# B&R Automation Studio project mappFramework (part 12)

#### variables.var - Name the suite and add PVs for the program
```iecst
(********************************************************************
 * COPYRIGHT --
 ********************************************************************
 * Program: utTemplate_automated
 * File: variables.var
 * Author: -
 * Created: -
 ********************************************************************
 * Local variables of program utTemplate_automated
 ********************************************************************)
(*Describe the test*)
VAR
	Testsuite : UtMgrTestSuite := (Name:='RecipeMgrVC4',Description:='RecipeMgr VC4 Unit Tests',MetaInformation:='Meta');
END_VAR
(*Variables used in the tests*)
VAR
	cycleCount : {REDUND_UNREPLICABLE} USINT;
	pMachineSettings : REFERENCE TO MachineSettingsType;
	MachineSettingsSize : {REDUND_UNREPLICABLE} UDINT;
	pParameters : REFERENCE TO ParametersType;
	ParameterSize : {REDUND_UNREPLICABLE} UDINT;
	LastSelectedIndex : UDINT;
	SetupState : USINT;
	FileName : STRING[24];
	NumberOfFiles : UINT;
	CurrentFile : UINT;
	fileInfo : fiDIR_READ_DATA;
	DirInfo_UT : DirInfo;
	DirRead_UT : DirRead;
	FileDelete_UT : FileDelete;
	FileCopy_UT : FileCopy;
END_VAR
```

#### testSuite.h
```c
#ifndef __TEST_SUITE_H__
#define __TEST_SUITE_H__

bool RecipeExists(char* recipeName);
bool SelectRecipe(char* wantedRecipe);
testStatusEnum RemoveNonDefaultFiles(USINT categoryIndex, char* selectFile, const char* category);

#endif
```

#### testSuite.c
```c
/********************************************************************
 * COPYRIGHT --
 ********************************************************************
 * Program: -
 * Author:
 * Created:
 ********************************************************************
 * Test registration and handshake
 ********************************************************************/

#include <bur/plctypes.h>

#ifdef _DEFAULT_INCLUDES
#include <AsDefault.h>
#endif

#include "UnitTest.h"
#include <string.h>
#include <stdbool.h>

void _INIT initTestSuite(void)
{
	Testsuite.Enable = 1;
	utInit(&Testsuite);

	CommonTestsuite.Enable = 1;
	utInit(&CommonTestsuite);

	strcpy((char*)&FileDeviceName, "mappRecipeFiles");
	strcpy((char*)&TextNameSpace, "mappFramework/Recipe/Alarms");
	strcpy((char*)&TextID, "SaveFailed");
	strcpy((char*)&HmiRecipe.Parameters.DeviceName, "mappRecipeFiles");

	PV_xgetadr("RecipeMgr:MachineSettings", (void*)&pMachineSettings, &MachineSettingsSize);
	PV_xgetadr("RecipeMgr:Parameters", (void*)&pParameters, &ParameterSize);

	LastSelectedIndex++;
}

void _CYCLIC cyclicWithTest(void)
{
	utCyclic(&Testsuite);
	if (Testsuite.Informational.LastKnownPassedLocation.TestCaseName != 0)
		strcpy((char*)&LastTestCase, (char*)Testsuite.Informational.LastKnownPassedLocation.TestCaseName);
	if (Testsuite.Informational.LastKnownPassedLocation.TestSetName != 0)
		strcpy((char*)&LastTestSet, (char*)Testsuite.Informational.LastKnownPassedLocation.TestSetName);
	if (Testsuite.Informational.LastKnownPassedLocation.File != 0)
		strcpy((char*)&LastTestFile, (char*)Testsuite.Informational.LastKnownPassedLocation.File);
}

void _EXIT exitTestSuite(void)
{
	utExit(&Testsuite);
}

bool RecipeExists(char* recipeName)
{
	for (USINT i = 0; i<(sizeof(MpRecipeUIConnect.Recipe.List.Names)/sizeof(MpRecipeUIConnect.Recipe.List.Names[0])); i++)
	{
		if (strcmp(recipeName, MpRecipeUIConnect.Recipe.List.Names[i]) == 0)
		{
			return true;
		}
	}
	return false;
}

bool SelectRecipe(char* wantedRecipe)
{
	if (((MpRecipeUIConnect.Status != mpRECIPE_UI_STATUS_IDLE) && (MpRecipeUIConnect.Status != mpRECIPE_UI_STATUS_ERROR)) &&
		(strcmp(wantedRecipe, HmiRecipe.Status.SelectedRecipe) != 0)) return false;

	for (USINT i=0; i <= MpRecipeUIConnect.Recipe.List.MaxSelection; i++)
	{
		if (strcmp(wantedRecipe, MpRecipeUIConnect.Recipe.List.Names[i]) == 0)
			MpRecipeUIConnect.Recipe.List.SelectedIndex = i;
	}

	return (strcmp(wantedRecipe, HmiRecipe.Status.SelectedRecipe) == 0);
}

testStatusEnum RemoveNonDefaultFiles(USINT categoryIndex, char* selectFile, const char* category)
{
	switch (SetupState)
	{
		case 0:
			DirInfo_UT.enable = true;
			DirInfo_UT.pDevice = (UDINT)&"mappRecipeFiles";
			DirInfo_UT.pPath = (UDINT)&"";
			DirInfo(&DirInfo_UT);
			TEST_BUSY_CONDITION(DirInfo_UT.status == 65535);
			TEST_ABORT_CONDITION(DirInfo_UT.status != 0);
			NumberOfFiles = DirInfo_UT.filenum;
			CurrentFile = 0;
			SetupState = (NumberOfFiles == 0) ? 100 : 1;
			break;

		case 1:
			DirRead_UT.enable = true;
			DirRead_UT.pDevice = DirInfo_UT.pDevice;
			DirRead_UT.entry = CurrentFile;
			DirRead_UT.option = fiFILE;
			DirRead_UT.pData = (UDINT)&fileInfo;
			DirRead_UT.data_len = sizeof(fileInfo);
			DirRead(&DirRead_UT);
			TEST_BUSY_CONDITION(DirRead_UT.status == 65535);
			TEST_ABORT_CONDITION(DirRead_UT.status != 0);
			SetupState = 2;
			break;

		case 2:
			if ((strcmp("Default.par", (char*)fileInfo.Filename) == 0) ||
				(strcmp("Machine.mcfg", (char*)fileInfo.Filename) == 0))
			{
				CurrentFile++;
				SetupState = (CurrentFile >= NumberOfFiles) ? 10 : 1;
				break;
			}
			FileDelete_UT.enable = true;
			FileDelete_UT.pDevice = DirInfo_UT.pDevice;
			FileDelete_UT.pName = (UDINT)&fileInfo.Filename;
			FileDelete(&FileDelete_UT);
			TEST_BUSY_CONDITION(FileDelete_UT.status == 65535);
			TEST_ABORT_CONDITION(FileDelete_UT.status != 0);

			NumberOfFiles--;
			SetupState = (CurrentFile >= NumberOfFiles) ? 10 : 1;
			break;

		case 10:
			strcpy((char*)&HmiRecipe.Parameters.DeviceName, "mappRecipeFiles");
			HmiRecipe.Parameters.CategoryIndex = categoryIndex;
			MpRecipeUIConnect.Recipe.Refresh = true;
			TEST_BUSY_CONDITION(MpRecipeUIConnect.Status != mpRECIPE_UI_STATUS_REFRESH)
			MpRecipeUIConnect.Recipe.Refresh = false;
			SetupState = 11;
			break;

		case 11:
			TEST_BUSY_CONDITION(MpRecipeUIConnect.Status != mpRECIPE_UI_STATUS_IDLE)
			TEST_BUSY_CONDITION(!RecipeExists(selectFile));
			TEST_BUSY_CONDITION(HmiRecipe.Status.HMIcommand != REC_HMI_WAIT)
			TEST_ABORT_CONDITION(pParameters == NULL);
			SetupState = 100;
			break;

		case 100:
			cycleCount = 0;
			TestState = TEST_ARRANGE;
			SetupState = 0;
			TEST_DONE;
	}
	TEST_BUSY;
}
```

#### Set_RecipeParameters.c
```c
#include <bur/plctypes.h>

#ifdef _DEFAULT_INCLUDES
#include <AsDefault.h>
#endif

#include "UnitTest.h"
#include <stdbool.h>
#include <string.h>
#include <stdlib.h>
#include "testSuite.h"

#define TIMEOUT_TEST_CASE									\
	if (cycleCount >= 254)									\
	{														\
		char abortMessage[80];								\
		char substate[10];									\
		memset(abortMessage, 0, sizeof(abortMessage));		\
		memset(substate, 0, sizeof(substate));				\
		itoa(ActSubState, substate, 10);					\
		strcpy(abortMessage, "Timeout in ActSubState = ");	\
		strcat(abortMessage, substate);						\
		TEST_FAIL(abortMessage);							\
		TEST_DONE;											\
	}

_SETUP_SET(void)
{
	return RemoveNonDefaultFiles(PARAMETERS_CATEGORY_INDEX, "Default.par", PARAMETERS_CATEGORY);
}

_TEARDOWN_SET(void)
{
	SetupState = 0;
	TEST_DONE;
}

_SETUP_TEST(void)
{
	ArrangeSubState = 0;
	ActSubState = 0;
	AssertSubState = 0;
	return RemoveNonDefaultFiles(PARAMETERS_CATEGORY_INDEX, "Default.par", PARAMETERS_CATEGORY);
}

_TEARDOWN_TEST(void)
{
	memset(&HmiRecipe.Commands, 0, sizeof(HmiRecipe.Commands));
	MpRecipeUIConnect.Recipe.Load = false;
	TEST_BUSY_CONDITION(!SelectRecipe("Default.par"));

	if (MpRecipeUIConnect.Status == mpRECIPE_UI_STATUS_ERROR)
	{
		MpRecipeUIConnect.Recipe.Refresh = true;
	}
	TEST_BUSY_CONDITION(MpRecipeUIConnect.Status != mpRECIPE_UI_STATUS_IDLE)
	MpRecipeUIConnect.Recipe.Refresh = false;

	TEST_DONE;
}

_CYCLIC_SET(void)
{
	cycleCount++;
}

_TEST DefaultValues(void)
{
	TIMEOUT_TEST_CASE
	switch (TestState)
	{
		case TEST_ARRANGE:
			// set MachineSettings through the pointer
			memset(pParameters, 0, sizeof(*pParameters));
			TEST_BUSY_CONDITION(!SelectRecipe("Default.par"));
			TEST_BUSY_CONDITION(MpRecipeUIConnect.Status != mpRECIPE_UI_STATUS_IDLE);
			TEST_BUSY_CONDITION(HmiRecipe.Status.HMIcommand != REC_HMI_WAIT);
			TestState = TEST_ACT;
			break;

		case TEST_ACT:
			switch (ActSubState)
			{
				case 0:
					MpRecipeUIConnect.Recipe.Load = true;
					TEST_BUSY_CONDITION(MpRecipeUIConnect.Status != mpRECIPE_UI_STATUS_LOAD);
					MpRecipeUIConnect.Recipe.Load = false;
					ActSubState = 1;
					break;

				case 1:
					TEST_BUSY_CONDITION(MpRecipeUIConnect.Status != mpRECIPE_UI_STATUS_IDLE);
					HmiRecipe.Commands.LoadRecipe = true;
					TEST_BUSY_CONDITION(HmiRecipe.Status.ProductRecipeLoaded == true);
					TEST_BUSY_CONDITION(HmiRecipe.Status.HMIcommand == REC_HMI_WAIT);
					HmiRecipe.Commands.LoadRecipe = false;
					ActSubState = 2;
					break;

				case 2:
					TEST_BUSY_CONDITION(HmiRecipe.Status.ProductRecipeLoaded == false);
					TEST_BUSY_CONDITION(HmiRecipe.Status.HMIcommand != REC_HMI_WAIT);
					TestState = TEST_ASSERT;
					break;
			}
			break;

		case TEST_ASSERT:
			TEST_ASSERT(Parameters.AddParametersHere1);
			TEST_ASSERT_EQUAL_STRING("two", Parameters.AddParametersHere2);
			TEST_ASSERT_DOUBLE_WITHIN(0.0001, 3.3, Parameters.AddParametersHere3);
			TEST_ASSERT_DOUBLE_WITHIN(0.0001, 4.4, Parameters.AddParametersHere4);
			TEST_ASSERT_DOUBLE_WITHIN(0.0001, 5.5, Parameters.AddParametersHere5);
			TEST_DONE;
			break;
	}
	TEST_BUSY;
}

_TEST CreateNew(void)
{
	TIMEOUT_TEST_CASE
	switch (TestState)
	{
		case TEST_ARRANGE:
			strcpy(HmiRecipe.Parameters.FileName, "test");
			TEST_BUSY_CONDITION(MpRecipeUIConnect.Status != mpRECIPE_UI_STATUS_IDLE);
			TEST_BUSY_CONDITION(HmiRecipe.Status.HMIcommand != REC_HMI_WAIT);
			TestState = TEST_ACT;
			break;

		case TEST_ACT:
			if (MpRecipeUIConnect.Status == mpRECIPE_UI_STATUS_ERROR)
			{
				TEST_FAIL("MpRecipeUIConnect in error state");
			}
			switch (ActSubState)
			{
				case 0:
					HmiRecipe.Commands.CreateRecipe = true;
					TEST_BUSY_CONDITION(MpRecipeUIConnect.Status != mpRECIPE_UI_STATUS_CREATE);
					HmiRecipe.Commands.CreateRecipe = false;
					ActSubState = 1;
					break;

				case 1:
					TEST_BUSY_CONDITION(MpRecipeUIConnect.Status != mpRECIPE_UI_STATUS_IDLE);
					TEST_BUSY_CONDITION(HmiRecipe.Status.ProductRecipeLoaded == false);
					ActSubState = 2;
					break;

				case 2:
					TEST_BUSY_CONDITION(MpRecipeUIConnect.Status == mpRECIPE_UI_STATUS_REFRESH);
					ActSubState = 3;
					break;

				case 3:
					TEST_BUSY_CONDITION(MpRecipeUIConnect.Status != mpRECIPE_UI_STATUS_IDLE);
					TestState = TEST_ASSERT;
					break;
			}
			break;

		case TEST_ASSERT:
			TEST_ASSERT(RecipeExists("test.par"));
			TEST_DONE;
			break;
	}

	TEST_BUSY;
}

_TEST CreateExisting(void)
{
	TIMEOUT_TEST_CASE
	switch (TestState)
	{
		case TEST_ARRANGE:
			strcpy(HmiRecipe.Parameters.FileName, "Default");
			TEST_BUSY_CONDITION(MpRecipeUIConnect.Status != mpRECIPE_UI_STATUS_IDLE);
			TEST_BUSY_CONDITION(HmiRecipe.Status.HMIcommand != REC_HMI_WAIT);
			TestState = TEST_ACT;
			break;

		case TEST_ACT:
			TestState = TEST_ASSERT;
			break;

		case TEST_ASSERT:
			HmiRecipe.Commands.CreateRecipe = false;
			TEST_ASSERT(HmiRecipe.Status.FileDuplicate);
			TEST_ASSERT(RecipeExists("Default.par"));
			TEST_DONE;
			break;
	}

	TEST_BUSY;
}

_TEST CreateNonExisting(void)
{
	TIMEOUT_TEST_CASE

	switch (TestState)
	{
		case TEST_ARRANGE:
			strcpy(HmiRecipe.Parameters.FileName, "test2");
			TEST_BUSY_CONDITION(MpRecipeUIConnect.Status != mpRECIPE_UI_STATUS_IDLE);
			TEST_BUSY_CONDITION(HmiRecipe.Status.HMIcommand != REC_HMI_WAIT);
			TestState = TEST_ACT;
			break;

		case TEST_ACT:
			TestState = TEST_ASSERT;
			break;

		case TEST_ASSERT:
			HmiRecipe.Commands.CreateRecipe = false;
			TEST_ASSERT(!HmiRecipe.Status.FileDuplicate);
			TEST_ASSERT(!RecipeExists("test2.par"));
			TEST_DONE;
			break;
	}
	TEST_BUSY;
}

_TEST CreateActive(void)
{
	TIMEOUT_TEST_CASE
	switch (TestState)
	{
		case TEST_ARRANGE:
			strcpy(HmiRecipe.Parameters.FileName, strtok(HmiRecipe.Status.LastLoadedProductRecipe, "."));
			TEST_BUSY_CONDITION(MpRecipeUIConnect.Status != mpRECIPE_UI_STATUS_IDLE);
			TEST_BUSY_CONDITION(HmiRecipe.Status.HMIcommand != REC_HMI_WAIT);
			TestState = TEST_ACT;
			break;

		case TEST_ACT:
			TestState = TEST_ASSERT;
			break;

		case TEST_ASSERT:
			HmiRecipe.Commands.CreateRecipe = false;
			TEST_ASSERT(HmiRecipe.Status.FileDuplicate);
			TEST_ASSERT(RecipeExists(HmiRecipe.Status.LastLoadedProductRecipe));
			TEST_DONE;
			break;
	}
	TEST_BUSY;
}

_TEST PreviewShouldNotAffectActive(void)
{
	TIMEOUT_TEST_CASE
	switch (TestState)
	{
		case TEST_ARRANGE:
			ParametersEdit.AddParametersHere1 = false;
			strcpy(ParametersEdit.AddParametersHere2, "testing preview");
			ParametersEdit.AddParametersHere3 = 12.56;
			ParametersEdit.AddParametersHere4 = 134.876;
			ParametersEdit.AddParametersHere5 = 87.4567;
			strcpy(HmiRecipe.Parameters.FileName, "preview");
			TEST_BUSY_CONDITION(MpRecipeUIConnect.Status != mpRECIPE_UI_STATUS_IDLE);
			TEST_BUSY_CONDITION(HmiRecipe.Status.HMIcommand != REC_HMI_WAIT);
			TestState = TEST_ACT;
			break;

		case TEST_ACT:
			if (MpRecipeUIConnect.Status == mpRECIPE_UI_STATUS_ERROR)
			{
				TEST_FAIL("MpRecipeUIConnect in error state");
				TEST_DONE;
			}
			switch (ActSubState)
			{
				case 0:
					HmiRecipe.Commands.CreateRecipe = true;
					TEST_BUSY_CONDITION(MpRecipeUIConnect.Status != mpRECIPE_UI_STATUS_CREATE);
					HmiRecipe.Commands.CreateRecipe = false;
					ActSubState = 1;
					break;

				case 1:
					TEST_BUSY_CONDITION(MpRecipeUIConnect.Status != mpRECIPE_UI_STATUS_IDLE);
					TEST_BUSY_CONDITION(HmiRecipe.Status.ProductRecipeLoaded == false);
					ActSubState = 2;
					break;

				case 2:
					TEST_BUSY_CONDITION(MpRecipeUIConnect.Status == mpRECIPE_UI_STATUS_REFRESH);
					ActSubState = 3;
					break;

				case 3:
					TEST_BUSY_CONDITION(MpRecipeUIConnect.Status != mpRECIPE_UI_STATUS_IDLE);
					TEST_BUSY_CONDITION(!SelectRecipe("preview.par"));
					ActSubState = 4;
					break;

				case 4:
					TEST_BUSY_CONDITION(MpRecipeSys.Load == true);
					TEST_BUSY_CONDITION(!SelectRecipe("preview.par"));
					MpRecipeUIConnect.Recipe.Load = true;
					TEST_BUSY_CONDITION(MpRecipeUIConnect.Status != mpRECIPE_UI_STATUS_LOAD);
					MpRecipeUIConnect.Recipe.Load = false;
					ActSubState = 5;
					break;

				case 5:
					TEST_BUSY_CONDITION(MpRecipeUIConnect.Status != mpRECIPE_UI_STATUS_IDLE);
					TestState = TEST_ASSERT;
					break;
			}
			break;

		case TEST_ASSERT:
			// check if preview affects the active parameters
			TEST_ASSERT(Parameters.AddParametersHere1);
			TEST_ASSERT_EQUAL_STRING("two", Parameters.AddParametersHere2);
			TEST_ASSERT_DOUBLE_WITHIN(0.0001, 3.3, Parameters.AddParametersHere3);
			TEST_ASSERT_DOUBLE_WITHIN(0.0001, 4.4, Parameters.AddParametersHere4);
			TEST_ASSERT_DOUBLE_WITHIN(0.0001, 5.5, Parameters.AddParametersHere5);
			TEST_DONE;
			break;
	}
	TEST_BUSY;
}

_TEST Preview(void)
{
	TIMEOUT_TEST_CASE

	switch (TestState)
	{
		case TEST_ARRANGE:
			ParametersEdit.AddParametersHere1 = false;
			strcpy(ParametersEdit.AddParametersHere2, "testing preview");
			ParametersEdit.AddParametersHere3 = 12.56;
			ParametersEdit.AddParametersHere4 = 134.876;
			ParametersEdit.AddParametersHere5 = 87.4567;
			strcpy(HmiRecipe.Parameters.FileName, "preview");
			TEST_BUSY_CONDITION(MpRecipeUIConnect.Status != mpRECIPE_UI_STATUS_IDLE);
			TEST_BUSY_CONDITION(HmiRecipe.Status.HMIcommand != REC_HMI_WAIT);
			TestState = TEST_ACT;
			break;

		case TEST_ACT:
			if (MpRecipeUIConnect.Status == mpRECIPE_UI_STATUS_ERROR)
			{
				TEST_FAIL("MpRecipeUIConnect in error state");
				TEST_DONE;
			}
			switch (ActSubState)
			{
				case 0:
					HmiRecipe.Commands.CreateRecipe = true;
					TEST_BUSY_CONDITION(MpRecipeUIConnect.Status != mpRECIPE_UI_STATUS_CREATE);
					HmiRecipe.Commands.CreateRecipe = false;
					ActSubState = 1;
					break;

				case 1:
					TEST_BUSY_CONDITION(MpRecipeUIConnect.Status != mpRECIPE_UI_STATUS_IDLE);
					TEST_BUSY_CONDITION(HmiRecipe.Status.ProductRecipeLoaded == false);
					ActSubState = 2;
					break;

				case 2:
					TEST_BUSY_CONDITION(MpRecipeUIConnect.Status == mpRECIPE_UI_STATUS_REFRESH);
					ActSubState = 3;
					break;

				case 3:
					TEST_BUSY_CONDITION(MpRecipeUIConnect.Status != mpRECIPE_UI_STATUS_IDLE);
					TEST_BUSY_CONDITION(!SelectRecipe("preview.par"));
					ActSubState = 4;
					break;

				case 4:
					TEST_BUSY_CONDITION(MpRecipeSys.Load == true);
					TEST_BUSY_CONDITION(!SelectRecipe("preview.par"));
					MpRecipeUIConnect.Recipe.Load = true;
					TEST_BUSY_CONDITION(MpRecipeUIConnect.Status != mpRECIPE_UI_STATUS_LOAD);
					MpRecipeUIConnect.Recipe.Load = false;
					ActSubState = 5;
					break;

				case 5:
					TEST_BUSY_CONDITION(MpRecipeUIConnect.Status != mpRECIPE_UI_STATUS_IDLE);
					TestState = TEST_ASSERT;
					break;
			}
			break;

		case TEST_ASSERT:
			TEST_ASSERT(!ParametersPreview.AddParametersHere1);
			TEST_ASSERT_EQUAL_STRING("testing preview", ParametersPreview.AddParametersHere2);
			TEST_ASSERT_DOUBLE_WITHIN(0.0001, 12.56, ParametersPreview.AddParametersHere3);
			TEST_ASSERT_DOUBLE_WITHIN(0.0001, 134.876, ParametersPreview.AddParametersHere4);
			TEST_ASSERT_DOUBLE_WITHIN(0.0001, 87.4567, ParametersPreview.AddParametersHere5);

			TEST_DONE;
			break;
	}
	TEST_BUSY;
}

_TEST Delete(void)
{
	TIMEOUT_TEST_CASE
	switch (TestState)
	{
		case TEST_ARRANGE:
			switch (ArrangeSubState)
			{
				case 0:
					strcpy(HmiRecipe.Parameters.FileName, "test");
					TEST_BUSY_CONDITION(MpRecipeUIConnect.Status != mpRECIPE_UI_STATUS_IDLE);
					TEST_BUSY_CONDITION(HmiRecipe.Status.HMIcommand != REC_HMI_WAIT);
					ArrangeSubState = 1;
					break;

				case 1:
					HmiRecipe.Commands.CreateRecipe = true;
					TEST_BUSY_CONDITION(MpRecipeUIConnect.Status != mpRECIPE_UI_STATUS_CREATE);
					HmiRecipe.Commands.CreateRecipe = false;
					ArrangeSubState = 2;
					break;

				case 2:
					TEST_BUSY_CONDITION(MpRecipeUIConnect.Status != mpRECIPE_UI_STATUS_IDLE);
					TEST_BUSY_CONDITION(HmiRecipe.Status.ProductRecipeLoaded == false);
					ArrangeSubState = 3;
					break;

				case 3:
					TEST_BUSY_CONDITION(MpRecipeUIConnect.Status == mpRECIPE_UI_STATUS_REFRESH);
					ArrangeSubState = 4;
					break;

				case 4:
					TEST_BUSY_CONDITION(MpRecipeUIConnect.Status != mpRECIPE_UI_STATUS_IDLE);
					ArrangeSubState = 5;
					break;

				case 5:
					TEST_BUSY_CONDITION(!SelectRecipe("test.par"));
					TEST_BUSY_CONDITION(MpRecipeUIConnect.Status != mpRECIPE_UI_STATUS_IDLE);
					TEST_BUSY_CONDITION(HmiRecipe.Status.HMIcommand != REC_HMI_WAIT);
					TestState = TEST_ACT;
					break;
			}
			break;

		case TEST_ACT:
			if (MpRecipeUIConnect.Status == mpRECIPE_UI_STATUS_ERROR)
			{
				TEST_FAIL("MpRecipeUIConnect in error state");
				TEST_DONE;
			}
			switch (ActSubState) {
				case 0:
					MpRecipeUIConnect.Recipe.Delete = true;
					TEST_BUSY_CONDITION(MpRecipeUIConnect.MessageBox.LayerStatus != 0);
					MpRecipeUIConnect.Recipe.Delete = false;
					MpRecipeUIConnect.MessageBox.Confirm = true;
					ActSubState = 1;
					break;

				case 1:
					MpRecipeUIConnect.MessageBox.Confirm = false;
					TEST_BUSY_CONDITION(MpRecipeUIConnect.MessageBox.LayerStatus == 0)
					TEST_BUSY_CONDITION(MpRecipeUIConnect.Status == mpRECIPE_UI_STATUS_IDLE);
					ActSubState = 2;
					break;

				case 2:
					TEST_BUSY_CONDITION(MpRecipeUIConnect.Status != mpRECIPE_UI_STATUS_IDLE);
					ActSubState = 3;
					break;

				case 3:
					TEST_BUSY_CONDITION(MpRecipeUIConnect.Status == mpRECIPE_UI_STATUS_REFRESH);
					ActSubState = 4;
					break;

				case 4:
					TEST_BUSY_CONDITION(MpRecipeUIConnect.Status != mpRECIPE_UI_STATUS_IDLE);
					TestState = TEST_ASSERT;
					break;
			}
			break;

		case TEST_ASSERT:
			TEST_ASSERT(!RecipeExists("test.par"));
			TEST_DONE;
			break;
	}
	TEST_BUSY;
}

_TEST Invalid(void)
{
	TIMEOUT_TEST_CASE
	switch (TestState)
	{
		case TEST_ARRANGE:
			switch (ArrangeSubState) {
				case 0:
					FileCopy_UT.enable = true;
					FileCopy_UT.pSrcDev = "mappRecipeFiles";
					FileCopy_UT.pSrc = "CSVformat\\Default.par";
					FileCopy_UT.pDestDev = "mappRecipeFiles";
					FileCopy_UT.pDest = "Invalid.par";
					FileCopy_UT.option= fiOVERWRITE;
					FileCopy(&FileCopy_UT);
					TEST_BUSY_CONDITION(FileCopy_UT.status == 65535);
					FileCopy_UT.enable = false;
					FileCopy(&FileCopy_UT);
					ArrangeSubState = 1;
					break;

				case 1:
					MpRecipeUIConnect.Recipe.Refresh = true;
					TEST_BUSY_CONDITION(MpRecipeUIConnect.Status == mpRECIPE_UI_STATUS_IDLE);
					MpRecipeUIConnect.Recipe.Refresh = false;
					ArrangeSubState = 2;
					break;

				case 2:
					TEST_BUSY_CONDITION(MpRecipeUIConnect.Status == mpRECIPE_UI_STATUS_REFRESH);
					ArrangeSubState = 3;
					break;

				case 3:
					TEST_BUSY_CONDITION(!SelectRecipe("Invalid.par"));
					TEST_BUSY_CONDITION(MpRecipeUIConnect.Status != mpRECIPE_UI_STATUS_IDLE);
					TEST_BUSY_CONDITION(HmiRecipe.Status.HMIcommand != REC_HMI_WAIT);
					TestState = TEST_ACT;
					break;
			}
			break;

		case TEST_ACT:
			switch (ActSubState)
			{
				case 0:
					MpRecipeUIConnect.Recipe.Load = true;
					TEST_BUSY_CONDITION(MpRecipeUIConnect.Status != mpRECIPE_UI_STATUS_LOAD);
					MpRecipeUIConnect.Recipe.Load = false;
					ActSubState = 1;
					break;

				case 1:
					TEST_BUSY_CONDITION(MpRecipeUIConnect.Status == mpRECIPE_UI_STATUS_LOAD);
					TestState = TEST_ASSERT;
					break;
			}
			break;

		case TEST_ASSERT:
			TEST_ASSERT_EQUAL_INT(mpRECIPE_UI_STATUS_ERROR, MpRecipeUIConnect.Status);
			TEST_DONE;
			break;
	}
	TEST_BUSY;
}

SKIP_TEST EditActive(void)
{
	TIMEOUT_TEST_CASE
	switch (TestState)
	{
		case TEST_ARRANGE:
			TEST_BUSY_CONDITION(!SelectRecipe("Default.par"));
			LastSelectedIndex++;
			TEST_BUSY_CONDITION(HmiRecipe.Status.HMIcommand != REC_HMI_WAIT);
			TEST_BUSY_CONDITION(MpRecipeUIConnect.Status != mpRECIPE_UI_STATUS_IDLE);

			ParametersEdit.AddParametersHere1 = false;
			strcpy(ParametersEdit.AddParametersHere2, "testing editing active");
			ParametersEdit.AddParametersHere3 = 12.56;
			ParametersEdit.AddParametersHere4 = 134.876;
			ParametersEdit.AddParametersHere5 = 87.4567;
			strcpy(HmiRecipe.Parameters.FileName, "editActive");
			TestState = TEST_ACT;
			break;

		case TEST_ACT:
			if (MpRecipeUIConnect.Status == mpRECIPE_UI_STATUS_ERROR)
			{
				TEST_FAIL("MpRecipeUIConnect in error state");
				TEST_DONE;
			}
			switch (ActSubState)
			{
				case 0:
					HmiRecipe.Commands.CreateRecipe = true;
					TEST_BUSY_CONDITION(MpRecipeUIConnect.Status != mpRECIPE_UI_STATUS_CREATE);
					HmiRecipe.Commands.CreateRecipe = false;
					ActSubState = 1;
					break;

				case 1:
					TEST_BUSY_CONDITION(MpRecipeUIConnect.Status != mpRECIPE_UI_STATUS_IDLE);
					TEST_BUSY_CONDITION(HmiRecipe.Status.ProductRecipeLoaded == false);
					ActSubState = 2;
					break;

				case 2:
					TEST_BUSY_CONDITION(MpRecipeUIConnect.Status == mpRECIPE_UI_STATUS_REFRESH);
					ActSubState = 3;
					break;

				case 3:
					TEST_BUSY_CONDITION(MpRecipeUIConnect.Status != mpRECIPE_UI_STATUS_IDLE);
					TEST_BUSY_CONDITION(HmiRecipe.Status.ProductRecipeLoaded == false);
					TEST_BUSY_CONDITION(!SelectRecipe("editActive.par"));
					ActSubState = 4;
					break;

				case 4:
					MpRecipeUIConnect.Recipe.Load = true;
					TEST_BUSY_CONDITION(MpRecipeUIConnect.Status != mpRECIPE_UI_STATUS_LOAD);
					MpRecipeUIConnect.Recipe.Load = false;
					ActSubState = 5;
					break;

				case 5:
					TEST_BUSY_CONDITION(MpRecipeUIConnect.Status != mpRECIPE_UI_STATUS_IDLE);
					ParametersEdit.AddParametersHere1 = true;
					strcpy(ParametersEdit.AddParametersHere2, "edited active");
					ParametersEdit.AddParametersHere3 = 52.56;
					ParametersEdit.AddParametersHere4 = 184.876;
					ParametersEdit.AddParametersHere5 = 587.4567;
					ActSubState = 6;
					break;

				case 6:
					HmiRecipe.Commands.SaveSelectedRecipe = true;
					TEST_BUSY_CONDITION(HmiRecipe.Status.HMIcommand == REC_HMI_WAIT);
					HmiRecipe.Commands.SaveSelectedRecipe = false;
					ActSubState = 7;
					break;

				case 7:
					TEST_BUSY_CONDITION(HmiRecipe.Status.HMIcommand != REC_HMI_WAIT);
					TEST_BUSY_CONDITION(MpRecipeUIConnect.Status != mpRECIPE_UI_STATUS_IDLE);
					TestState = TEST_ASSERT;
					break;
			}
			break;

		case TEST_ASSERT:
			TEST_ASSERT(Parameters.AddParametersHere1);
			TEST_ASSERT_EQUAL_STRING("edited active", Parameters.AddParametersHere2);
			TEST_ASSERT_DOUBLE_WITHIN(0.0001, 52.56, Parameters.AddParametersHere3);
			TEST_ASSERT_DOUBLE_WITHIN(0.0001, 184.876, Parameters.AddParametersHere4);
			TEST_ASSERT_DOUBLE_WITHIN(0.0001, 587.4567, Parameters.AddParametersHere5);

			TEST_DONE;
			break;
	}
	TEST_BUSY;
}

/*
B+R UnitTest: This is generated code.
Do not edit! Do not move!
Description: UnitTest Testprogramm infrastructure (TestSet).
LastUpdated: 2023-08-25 18:59:10Z
By B+R UnitTest Helper Version: 2.0.1.59
*/
UNITTEST_FIXTURES(fixtures)
{
	new_TestFixture("DefaultValues", DefaultValues),
	new_TestFixture("CreateNew", CreateNew),
	new_TestFixture("CreateExisting", CreateExisting),
	new_TestFixture("CreateNonExisting", CreateNonExisting),
	new_TestFixture("CreateActive", CreateActive),
	new_TestFixture("PreviewShouldNotAffectActive", PreviewShouldNotAffectActive),
	new_TestFixture("Preview", Preview),
	new_TestFixture("Delete", Delete),
	new_TestFixture("Invalid", Invalid),
	skipTestFixture("EditActive", EditActive),
};

UNITTEST_CALLER_COMPLETE_EXPLICIT(Set_RecipeParameters, "Set_RecipeParameters", setupTest, teardownTest, fixtures, setupSet, teardownSet, cyclicSetCaller);
```

#### Set_RecipeMachineSettings.c
```c
#include <bur/plctypes.h>

#ifdef _DEFAULT_INCLUDES
#include <AsDefault.h>
#endif

#include "UnitTest.h"
#include <stdbool.h>
#include <string.h>
#include <stdlib.h>
#include "testSuite.h"

#define TIMEOUT_TEST_CASE									\
	if (cycleCount >= 254)									\
	{														\
		char abortMessage[80];								\
		char substate[10];									\
		memset(abortMessage, 0, sizeof(abortMessage));		\
		memset(substate, 0, sizeof(substate));				\
		itoa(ActSubState, substate, 10);					\
		strcpy(abortMessage, "Timeout in ActSubState = ");	\
		strcat(abortMessage, substate);						\
		TEST_FAIL(abortMessage);							\
		TEST_DONE;											\
	}

_SETUP_SET(void)
{
	return RemoveNonDefaultFiles(MACH_CONFIG_CATEGORY_INDEX, "Machine.mcfg", MACHINE_CONFIGURATION_CATEGORY);
}

_TEARDOWN_SET(void)
{
	SetupState = 0;
	TEST_DONE;
}

_SETUP_TEST(void)
{
	ArrangeSubState = 0;
	ActSubState = 0;
	AssertSubState = 0;
	return RemoveNonDefaultFiles(MACH_CONFIG_CATEGORY_INDEX, "Machine.mcfg", MACHINE_CONFIGURATION_CATEGORY);
}

_TEARDOWN_TEST(void)
{
	memset(&HmiRecipe.Commands, 0, sizeof(HmiRecipe.Commands));
	MpRecipeUIConnect.Recipe.Load = false;
	TEST_BUSY_CONDITION(!SelectRecipe("Machine.mcfg"));

	if (MpRecipeUIConnect.Status == mpRECIPE_UI_STATUS_ERROR)
	{
		MpRecipeUIConnect.Recipe.Refresh = true;
	}
	TEST_BUSY_CONDITION(MpRecipeUIConnect.Status != mpRECIPE_UI_STATUS_IDLE)
	MpRecipeUIConnect.Recipe.Refresh = false;

	TEST_DONE;
}

_CYCLIC_SET(void)
{
	cycleCount++;
}

_TEST DefaultValues(void)
{
	TIMEOUT_TEST_CASE
	switch (TestState)
	{
		case TEST_ARRANGE:
			// set MachineSettings through the pointer
			memset(pMachineSettings, 0, sizeof(*pMachineSettings));
			TEST_BUSY_CONDITION(!SelectRecipe("Machine.mcfg"));
			TEST_BUSY_CONDITION(MpRecipeUIConnect.Status != mpRECIPE_UI_STATUS_IDLE);
			TEST_BUSY_CONDITION(HmiRecipe.Status.HMIcommand != REC_HMI_WAIT);
			TestState = TEST_ACT;
			break;

		case TEST_ACT:
			if (MpRecipeUIConnect.Status == mpRECIPE_UI_STATUS_ERROR)
			{
				TEST_FAIL("MpRecipeUIConnect in error state");
				TEST_DONE;
			}
			switch (ActSubState)
			{
				case 0:
					MpRecipeUIConnect.Recipe.Load = true;
					HmiRecipe.Commands.LoadRecipe = true;
					TEST_BUSY_CONDITION(HmiRecipe.Status.ConfigRecipeLoaded == true);
					TEST_BUSY_CONDITION(HmiRecipe.Status.HMIcommand == REC_HMI_WAIT);
					HmiRecipe.Commands.LoadRecipe = false;
					MpRecipeUIConnect.Recipe.Load = false;
					ActSubState = 1;
					break;
				case 1:
					TEST_BUSY_CONDITION(HmiRecipe.Status.ConfigRecipeLoaded == false);
					TEST_BUSY_CONDITION(HmiRecipe.Status.HMIcommand != REC_HMI_WAIT);
					TEST_BUSY_CONDITION(MpRecipeUIConnect.Status == mpRECIPE_UI_STATUS_LOAD);
					TestState = TEST_ASSERT;
					break;
			}
			break;

		case TEST_ASSERT:
			TEST_ASSERT_EQUAL_INT(11, MachineSettings.AddMachineSettingsHere1);
			TEST_ASSERT_EQUAL_INT(22, MachineSettings.AddMachineSettingsHere2);
			TEST_ASSERT_EQUAL_INT(true, MachineSettings.AddMachineSettingsHere3);
			TEST_ASSERT_DOUBLE_WITHIN(0.0001, 3.2999999, MachineSettings.AddMachineSettingsHere4);
			TEST_ASSERT_EQUAL_INT(44, MachineSettings.AddMachineSettingsHere5);
			TEST_DONE;
			break;
	}
	TEST_BUSY;

	TEST_DONE;
}
_TEST CreateNew(void)
{
	TIMEOUT_TEST_CASE
	switch (TestState)
	{
		case TEST_ARRANGE:
			strcpy(HmiRecipe.Parameters.FileName, "test");
			TEST_BUSY_CONDITION(MpRecipeUIConnect.Status != mpRECIPE_UI_STATUS_IDLE);
			TEST_BUSY_CONDITION(HmiRecipe.Status.HMIcommand != REC_HMI_WAIT);
			TestState = TEST_ACT;
			break;

		case TEST_ACT:
			if (MpRecipeUIConnect.Status == mpRECIPE_UI_STATUS_ERROR)
			{
				TEST_FAIL("MpRecipeUIConnect in error state");
				TEST_DONE;
			}
			switch (ActSubState)
			{
				case 0:
					HmiRecipe.Commands.CreateRecipe = true;
					TEST_BUSY_CONDITION(MpRecipeUIConnect.Status != mpRECIPE_UI_STATUS_CREATE);
					HmiRecipe.Commands.CreateRecipe = false;
					ActSubState = 1;
					break;

				case 1:
					TEST_BUSY_CONDITION(MpRecipeUIConnect.Status != mpRECIPE_UI_STATUS_IDLE);
					TEST_BUSY_CONDITION(HmiRecipe.Status.ProductRecipeLoaded == false);
					ActSubState = 2;
					break;

				case 2:
					TEST_BUSY_CONDITION(MpRecipeUIConnect.Status == mpRECIPE_UI_STATUS_REFRESH);
					ActSubState = 3;
					break;

				case 3:
					TEST_BUSY_CONDITION(MpRecipeUIConnect.Status != mpRECIPE_UI_STATUS_IDLE);
					TestState = TEST_ASSERT;
					break;
			}
			break;

		case TEST_ASSERT:
			TEST_ASSERT(RecipeExists("test.mcfg"));
			TEST_DONE;
			break;
	}
	TEST_BUSY;

}

_TEST CreateExisting(void)
{
	TIMEOUT_TEST_CASE
	switch (TestState)
	{
		case TEST_ARRANGE:
			strcpy(HmiRecipe.Parameters.FileName, "Machine");
			TEST_BUSY_CONDITION(MpRecipeUIConnect.Status != mpRECIPE_UI_STATUS_IDLE);
			TEST_BUSY_CONDITION(HmiRecipe.Status.HMIcommand != REC_HMI_WAIT);
			TestState = TEST_ACT;
			break;

		case TEST_ACT:
			TestState = TEST_ASSERT;
			break;

		case TEST_ASSERT:
			HmiRecipe.Commands.CreateRecipe = false;
			TEST_ASSERT(HmiRecipe.Status.FileDuplicate);
			TEST_ASSERT(RecipeExists("Machine.mcfg"));
			TEST_DONE;
			break;
	}
	TEST_BUSY;
}

_TEST CreateNonExisting(void)
{
	TIMEOUT_TEST_CASE
	switch (TestState)
	{
		case TEST_ARRANGE:
			strcpy(HmiRecipe.Parameters.FileName, "test2");
			TEST_BUSY_CONDITION(MpRecipeUIConnect.Status != mpRECIPE_UI_STATUS_IDLE);
			TEST_BUSY_CONDITION(HmiRecipe.Status.HMIcommand != REC_HMI_WAIT);
			TestState = TEST_ACT;
			break;

		case TEST_ACT:
			TestState = TEST_ASSERT;
			break;

		case TEST_ASSERT:
			HmiRecipe.Commands.CreateRecipe = false;
			TEST_ASSERT(!HmiRecipe.Status.FileDuplicate);
			TEST_ASSERT(!RecipeExists("test2.mcfg"));
			TEST_DONE;
			break;
	}
	TEST_BUSY;
}

_TEST CreateActive(void)
{
	TIMEOUT_TEST_CASE
	switch (TestState)
	{
		case TEST_ARRANGE:
			strcpy(HmiRecipe.Parameters.FileName, strtok(HmiRecipe.Status.LastLoadedConfigRecipe, "."));
			TEST_BUSY_CONDITION(MpRecipeUIConnect.Status != mpRECIPE_UI_STATUS_IDLE);
			TEST_BUSY_CONDITION(HmiRecipe.Status.HMIcommand != REC_HMI_WAIT);
			TestState = TEST_ACT;
			break;

		case TEST_ACT:
			TestState = TEST_ASSERT;
			break;

		case TEST_ASSERT:
			HmiRecipe.Commands.CreateRecipe = false;
			TEST_ASSERT(HmiRecipe.Status.FileDuplicate);
			TEST_ASSERT(RecipeExists(HmiRecipe.Status.LastLoadedConfigRecipe));
			TEST_DONE;
			break;
	}
	TEST_BUSY;
}

_TEST Preview(void)
{
	TIMEOUT_TEST_CASE
	switch (TestState)
	{
		case TEST_ARRANGE:
			MachineSettings.AddMachineSettingsHere1 = 157;
			MachineSettings.AddMachineSettingsHere2 = 43956;
			MachineSettings.AddMachineSettingsHere3 = true;
			MachineSettings.AddMachineSettingsHere4 = 134.876;
			MachineSettings.AddMachineSettingsHere5 = 4373;
			strcpy(HmiRecipe.Parameters.FileName, "preview");
			TEST_BUSY_CONDITION(MpRecipeUIConnect.Status != mpRECIPE_UI_STATUS_IDLE);
			TEST_BUSY_CONDITION(HmiRecipe.Status.HMIcommand != REC_HMI_WAIT);
			TestState = TEST_ACT;
			break;

		case TEST_ACT:
			if (MpRecipeUIConnect.Status == mpRECIPE_UI_STATUS_ERROR)
			{
				TEST_FAIL("MpRecipeUIConnect in error state");
				TEST_DONE;
			}
			switch (ActSubState)
			{
				case 0:
					HmiRecipe.Commands.CreateRecipe = true;
					TEST_BUSY_CONDITION(MpRecipeUIConnect.Status != mpRECIPE_UI_STATUS_CREATE);
					HmiRecipe.Commands.CreateRecipe = false;
					ActSubState = 1;
				break;

				case 1:
					TEST_BUSY_CONDITION(MpRecipeUIConnect.Status != mpRECIPE_UI_STATUS_IDLE);
					TEST_BUSY_CONDITION(HmiRecipe.Status.ProductRecipeLoaded == false);
					ActSubState = 2;
				break;

				case 2:
					TEST_BUSY_CONDITION(MpRecipeUIConnect.Status == mpRECIPE_UI_STATUS_REFRESH);
					ActSubState = 3;
				break;

				case 3:
					TEST_BUSY_CONDITION(MpRecipeUIConnect.Status != mpRECIPE_UI_STATUS_IDLE);
					TEST_BUSY_CONDITION(!SelectRecipe("preview.mcfg"));
					ActSubState = 4;
				break;

				case 4:
					TEST_BUSY_CONDITION(!SelectRecipe("preview.mcfg"));
					MpRecipeUIConnect.Recipe.Load = true;
					TEST_BUSY_CONDITION(MpRecipeUIConnect.Status != mpRECIPE_UI_STATUS_LOAD);
					MpRecipeUIConnect.Recipe.Load = false;
					ActSubState = 5;
				break;

				case 5:
					TEST_BUSY_CONDITION(MpRecipeUIConnect.Status != mpRECIPE_UI_STATUS_IDLE);
					TestState = TEST_ASSERT;
				break;
			}
			break;

		case TEST_ASSERT:
			TEST_ASSERT_EQUAL_INT(11, MachineSettings.AddMachineSettingsHere1);
			TEST_ASSERT_EQUAL_INT(22, MachineSettings.AddMachineSettingsHere2);
			TEST_ASSERT_EQUAL_INT(true, MachineSettings.AddMachineSettingsHere3);
			TEST_ASSERT_DOUBLE_WITHIN(0.0001, 3.2999999, MachineSettings.AddMachineSettingsHere4);
			TEST_ASSERT_EQUAL_INT(44, MachineSettings.AddMachineSettingsHere5);
			TEST_DONE;
			break;
	}
	TEST_BUSY;
}

_TEST Delete(void)
{
	TIMEOUT_TEST_CASE
	switch (TestState)
	{
		case TEST_ARRANGE:
			switch (ArrangeSubState)
			{
				case 0:
					strcpy(HmiRecipe.Parameters.FileName, "test");
					TEST_BUSY_CONDITION(MpRecipeUIConnect.Status != mpRECIPE_UI_STATUS_IDLE);
					TEST_BUSY_CONDITION(HmiRecipe.Status.HMIcommand != REC_HMI_WAIT);
					ArrangeSubState = 1;
					break;

				case 1:
					HmiRecipe.Commands.CreateRecipe = true;
					TEST_BUSY_CONDITION(MpRecipeUIConnect.Status != mpRECIPE_UI_STATUS_CREATE);
					HmiRecipe.Commands.CreateRecipe = false;
					ArrangeSubState = 2;
					break;

				case 2:
					TEST_BUSY_CONDITION(MpRecipeUIConnect.Status != mpRECIPE_UI_STATUS_IDLE);
					TEST_BUSY_CONDITION(HmiRecipe.Status.ProductRecipeLoaded == false);
					ArrangeSubState = 3;
					break;

				case 3:
					TEST_BUSY_CONDITION(MpRecipeUIConnect.Status == mpRECIPE_UI_STATUS_REFRESH);
					ArrangeSubState = 4;
					break;

				case 4:
					TEST_BUSY_CONDITION(MpRecipeUIConnect.Status != mpRECIPE_UI_STATUS_IDLE);
					ArrangeSubState = 5;
					break;

				case 5:
					TEST_BUSY_CONDITION(!SelectRecipe("test.mcfg"));
					TEST_BUSY_CONDITION(MpRecipeUIConnect.Status != mpRECIPE_UI_STATUS_IDLE);
					TEST_BUSY_CONDITION(HmiRecipe.Status.HMIcommand != REC_HMI_WAIT);
					TestState = TEST_ACT;
					break;
			}
			break;

		case TEST_ACT:
			if (MpRecipeUIConnect.Status == mpRECIPE_UI_STATUS_ERROR)
			{
				TEST_FAIL("MpRecipeUIConnect in error state");
				TEST_DONE;
			}
			switch (ActSubState)
			{
				case 0:
					MpRecipeUIConnect.Recipe.Delete = true;
					TEST_BUSY_CONDITION(MpRecipeUIConnect.MessageBox.LayerStatus != 0);
					MpRecipeUIConnect.Recipe.Delete = false;
					MpRecipeUIConnect.MessageBox.Confirm = true;
					ActSubState = 1;
					break;

				case 1:
					MpRecipeUIConnect.MessageBox.Confirm = false;
					TEST_BUSY_CONDITION(MpRecipeUIConnect.MessageBox.LayerStatus == 0)
					TEST_BUSY_CONDITION(MpRecipeUIConnect.Status == mpRECIPE_UI_STATUS_IDLE);
					ActSubState = 2;
					break;

				case 2:
					TEST_BUSY_CONDITION(MpRecipeUIConnect.Status != mpRECIPE_UI_STATUS_IDLE);
					ActSubState = 3;
					break;

				case 3:
					TEST_BUSY_CONDITION(MpRecipeUIConnect.Status == mpRECIPE_UI_STATUS_REFRESH);
					ActSubState = 4;
					break;

				case 4:
					TEST_BUSY_CONDITION(MpRecipeUIConnect.Status != mpRECIPE_UI_STATUS_IDLE);
					TestState = TEST_ASSERT;
					break;
			}
			break;

		case TEST_ASSERT:
			TEST_ASSERT(!RecipeExists("test.mcfg"));
			TEST_DONE;
			break;
	}
	TEST_BUSY;
}

_TEST Invalid(void)
{
	TIMEOUT_TEST_CASE
	switch (TestState)
	{
		case TEST_ARRANGE:
			switch (ArrangeSubState) {
				case 0:
					FileCopy_UT.enable = true;
					FileCopy_UT.pSrcDev = "mappRecipeFiles";
					FileCopy_UT.pSrc = "CSVformat\\Machine.mcfg";
					FileCopy_UT.pDestDev = "mappRecipeFiles";
					FileCopy_UT.pDest = "MachineInvalid.mcfg";
					FileCopy_UT.option= fiOVERWRITE;
					FileCopy(&FileCopy_UT);
					TEST_BUSY_CONDITION(FileCopy_UT.status == 65535);
					FileCopy_UT.enable = false;
					FileCopy(&FileCopy_UT);
					ArrangeSubState = 1;
					break;

				case 1:
					MpRecipeUIConnect.Recipe.Refresh = true;
					TEST_BUSY_CONDITION(MpRecipeUIConnect.Status == mpRECIPE_UI_STATUS_IDLE);
					MpRecipeUIConnect.Recipe.Refresh = false;
					ArrangeSubState = 2;
					break;

				case 2:
					TEST_BUSY_CONDITION(MpRecipeUIConnect.Status == mpRECIPE_UI_STATUS_REFRESH);
					ArrangeSubState = 3;
					break;

				case 3:
					TEST_BUSY_CONDITION(!SelectRecipe("MachineInvalid.mcfg"));
					TEST_BUSY_CONDITION(MpRecipeUIConnect.Status != mpRECIPE_UI_STATUS_IDLE);
					TEST_BUSY_CONDITION(HmiRecipe.Status.HMIcommand != REC_HMI_WAIT);
					TestState = TEST_ACT;
					break;
			}
			break;

		case TEST_ACT:
			switch (ActSubState)
			{
				case 0:
					MpRecipeUIConnect.Recipe.Load = true;
					TEST_BUSY_CONDITION(MpRecipeUIConnect.Status != mpRECIPE_UI_STATUS_LOAD);
					MpRecipeUIConnect.Recipe.Load = false;
					ActSubState = 1;
					break;

				case 1:
					TEST_BUSY_CONDITION(MpRecipeUIConnect.Status == mpRECIPE_UI_STATUS_LOAD);
					TestState = TEST_ASSERT;
					break;
			}
			break;

		case TEST_ASSERT:
			TEST_ASSERT_EQUAL_INT(mpRECIPE_UI_STATUS_ERROR, MpRecipeUIConnect.Status);
			TEST_DONE;
			break;
	}
	TEST_BUSY;
}

/*
B+R UnitTest: This is generated code.
Do not edit! Do not move!
Description: UnitTest Testprogramm infrastructure (TestSet).
LastUpdated: 2023-08-25 18:59:10Z
By B+R UnitTest Helper Version: 2.0.1.59
*/
UNITTEST_FIXTURES(fixtures)
{
	new_TestFixture("DefaultValues", DefaultValues),
	new_TestFixture("CreateNew", CreateNew),
	new_TestFixture("CreateExisting", CreateExisting),
	new_TestFixture("CreateNonExisting", CreateNonExisting),
	new_TestFixture("CreateActive", CreateActive),
	new_TestFixture("Preview", Preview),
	new_TestFixture("Delete", Delete),
	new_TestFixture("Invalid", Invalid),
};

UNITTEST_CALLER_COMPLETE_EXPLICIT(Set_RecipeMachineSettings, "Set_RecipeMachineSettings", setupTest, teardownTest, fixtures, setupSet, teardownSet, cyclicSetCaller);
```

### Package Logical/UnitTestVC4/UserX - Package for mapp UserX Framework

### Program Logical/UnitTestVC4/UserX/UserXUnitTest (ANSIC)

- UserXMgr.typ (reference to Logical/Infrastructure/VC4/UserX/UserXMgr/UserXMgr.typ)

- UserXMgr.var (reference to Logical/Infrastructure/VC4/UserX/UserXMgr/UserXMgr.var)

#### variables.var - Name the suite and add PVs for the program
```iecst
(********************************************************************
 * COPYRIGHT --
 ********************************************************************
 * Program: utTemplate_automated
 * File: variables.var
 * Author: -
 * Created: -
 ********************************************************************
 * Local variables of program utTemplate_automated
 ********************************************************************)
(*Describe the test*)
VAR
	TestStep : USINT;
	Testsuite : UtMgrTestSuite := (Name:='UserMgrVC4',Description:='UserMgr VC4 Unit Tests',MetaInformation:='Meta');
END_VAR
(*Variables used in the tests*)
VAR
	cycleCount : USINT;
	UT_Password : WSTRING[80] := "123ABc"; (*Unit test password login request*)
	UT_Username : WSTRING[80] := "Admin"; (*Unit test username login request *)
	UT_Compare : DINT; (*Unit test string compare PV holder*)
	UT_Message : STRING[80]; (*Unit test message variable*)
	UT_j : USINT; (*index for FOR loops*)
	UT_i : USINT; (*index for FOR loops*)
	UT_RoleList : ARRAY[0..4] OF WSTRING[50] := ["Administrators","Operators","Service",2("")]; (*Unit test role list for checking against user list*)
	UT_UserList : ARRAY[0..4] OF WSTRING[50] := ["Admin","Operator","Service_Tech",2("")]; (*Unit test user list for checking against user list*)
END_VAR
```

#### testSuite.c
```c
/********************************************************************
 * COPYRIGHT --
 ********************************************************************
 * Program: -
 * Author:
 * Created:
 ********************************************************************
 * Test registration and handshake
 ********************************************************************/

#include <bur/plctypes.h>

#ifdef _DEFAULT_INCLUDES
#include <AsDefault.h>
#endif
#include <string.h>

#include "UnitTest.h"

void _INIT initTestSuite(void)
{
	Testsuite.Enable = 1;
	utInit(&Testsuite);

	CommonTestsuite.Enable = 1;
	utInit(&CommonTestsuite);

	strcpy((char*)&FileDeviceName, "mappUserXFiles");
	strcpy((char*)&TextNameSpace, "mappFramework/UserX/Alarms");
	strcpy((char*)&TextID, "UserLocked");

}

void _CYCLIC cyclicWithTest(void)
{
	utCyclic(&Testsuite);
}

void _EXIT exitTestSuite(void)
{
	utExit(&Testsuite);
}
```

- Set_Common.c (reference to Logical/UnitTestVC4/Common/CommonUT/Set_Common.c)

### Package Logical/UnitTestVC4/Report - Package for mapp Report Framework

### Program Logical/UnitTestVC4/Report/ReportUnitTest (ANSIC) - Unit Tests for ReportMgr

- ReportMgr.typ (reference to Logical/Infrastructure/VC4/Report/ReportMgr/ReportMgr.typ)

- ReportMgr.var (reference to Logical/Infrastructure/VC4/Report/ReportMgr/ReportMgr.var)

#### variables.var - Name the suite and add PVs for the program
```iecst
(********************************************************************
 * COPYRIGHT --
 ********************************************************************
 * Program: utTemplate_automated
 * File: variables.var
 * Author: -
 * Created: -
 ********************************************************************
 * Local variables of program utTemplate_automated
 ********************************************************************)
(*Describe the test*)
VAR
	Testsuite : UtMgrTestSuite := (Name:='ReportMgrVC4',Description:='ReportMgr VC4 Unit Tests',MetaInformation:='Meta');
END_VAR
(*Variables used in the tests*)
VAR
	HmiReport_UT : ReportHmiInterfaceType; (*HMI interface structure*)
	CoreInfo_UT : MpReportCoreInfoType;
	CoreInfoActive : BOOL;
	CoreCmdDone : BOOL;
END_VAR
```

#### Set_ReportMgr.c
```c
#include <bur/plctypes.h>

#ifdef _DEFAULT_INCLUDES
#include <AsDefault.h>
#endif

#include "UnitTest.h"
#include <stdbool.h>
#include <string.h>

_SETUP_SET(void)
{
	TEST_DONE;
}

_TEARDOWN_SET(void)
{
	TEST_DONE;
}

_SETUP_TEST(void)
{
	TEST_DONE;
}

_TEARDOWN_TEST(void)
{
	TEST_DONE;
}

_TEST CreateAdvReport(void)
{
	switch (TestState)
	{
		case TEST_ARRANGE:
			HmiReport_UT.Parameters.UseAdvancedFormat = true;
			TEST_BUSY_CONDITION(CoreInfoActive == true);
			TEST_ABORT_CONDITION(HmiReport_UT.Status.Error == true);
			TestState = TEST_ACT;
			break;

		case TEST_ACT:
			TEST_BUSY_CONDITION(CoreInfoActive == false);
			HmiReport_UT.Commands.Generate = true;
			TEST_BUSY_CONDITION(HmiReport_UT.Status.Busy == false);
			TestState = TEST_ASSERT;
			break;

		case TEST_ASSERT:
			HmiReport_UT.Commands.Generate = false;
			TEST_BUSY_CONDITION(HmiReport_UT.Status.Busy == true);
			TEST_ASSERT(HmiReport_UT.Status.Error == false);
			TEST_ASSERT_EQUAL_INT(1, CoreInfo_UT.NumberOfReports);
			TEST_DONE;
			break;
	}
	TEST_BUSY;
}

_TEST CreateSimpleReport(void)
{
	switch (TestState)
	{
		case TEST_ARRANGE:
			HmiReport_UT.Parameters.UseAdvancedFormat = false;
			TEST_BUSY_CONDITION(CoreInfoActive == true);
			TEST_ABORT_CONDITION(HmiReport_UT.Status.Error == true);
			TestState = TEST_ACT;
			break;

		case TEST_ACT:
			TEST_BUSY_CONDITION(CoreInfoActive == false);
			HmiReport_UT.Commands.Generate = true;
			TEST_BUSY_CONDITION(HmiReport_UT.Status.Busy == false);
			TestState = TEST_ASSERT;
			break;

		case TEST_ASSERT:
			HmiReport_UT.Commands.Generate = false;
			TEST_BUSY_CONDITION(HmiReport_UT.Status.Busy == true);
			TEST_ASSERT(HmiReport_UT.Status.Error == false);
			TEST_ASSERT_EQUAL_INT(1, CoreInfo_UT.NumberOfReports);
			TEST_DONE;
			break;
	}
	TEST_BUSY;
}

/*
B+R UnitTest: This is generated code.
Do not edit! Do not move!
Description: UnitTest Testprogramm infrastructure (TestSet).
LastUpdated: 2022-11-15 21:58:19Z
By B+R UnitTest Helper Version: 2.0.1.59
*/
UNITTEST_FIXTURES(fixtures)
{
	new_TestFixture("CreateAdvReport", CreateAdvReport),
	new_TestFixture("CreateSimpleReport", CreateSimpleReport),
};

UNITTEST_CALLER_COMPLETE_EXPLICIT(Set_ReportMgr, "Set_ReportMgr", setupTest, teardownTest, fixtures, setupSet, teardownSet, 0);
```

#### CommonTypes.typ
```iecst
TYPE
	TestCaseEnum :
		(
		TEST_ARRANGE,
		TEST_ACT,
		TEST_ASSERT
		);
END_TYPE
```

- Set_Common.c (reference to Logical/UnitTestVC4/Common/CommonUT/Set_Common.c)

### Program Logical/UnitTestVC4/Common/CommonUT (ANSIC)

- CommonTypes.typ (reference to Logical/UnitTestVC4/Common/CommonUT/CommonTypes.typ)

#### testSuite.c
```c
/********************************************************************
 * COPYRIGHT --
 ********************************************************************
 * Program: -
 * Author:
 * Created:
 ********************************************************************
 * Test registration and handshake
 ********************************************************************/

#include <bur/plctypes.h>

#ifdef _DEFAULT_INCLUDES
#include <AsDefault.h>
#endif

#include "UnitTest.h"

void _INIT initTestSuite(void)
{
	Testsuite.Enable = 1;
	utInit(&Testsuite);
}

void _CYCLIC cyclicWithTest(void)
{
	utCyclic(&Testsuite);
}

void _EXIT exitTestSuite(void)
{
	utExit(&Testsuite);
}
```

- Set_Common.c (reference to Logical/UnitTestVC4/Common/CommonUT/Set_Common.c)

- Visualisation Logical/VC4/mappFrameworkVisu (not shown)

Listed in the project but not available here: Logical/Global.typ, Logical/Global.var, Logical/Infrastructure/Backup/BackupMgr/ChangeConfiguration.st, Logical/Infrastructure/VC4/Audit/ExportedText, Logical/MachineControl/AxisTemplate/AxisMgr/LocalFunctions.fun, Logical/MachineControl/AppAxis_1/AppAxis_1/LocalFunctions.fun, Logical/MachineControl/AppAxis_1/AppAxis_1/AutomaticCommand.st, Logical/UserPartition/Recipe/CSVformat, Logical/UserPartition/Recipe/XMLformat, Logical/UnitTest/Libraries/UnitTest/UnitTest.h, Logical/UnitTest/Libraries/UnitTest/include/AssertImpl.h, Logical/UnitTest/Libraries/UnitTest/include/HelperMacro.h, Logical/UnitTest/Libraries/UnitTest/include/utRunner.h, Logical/UnitTest/Libraries/UnitTest/include/Test.h, Logical/UnitTest/Libraries/UnitTest/include/TestListener.h, Logical/UnitTest/Libraries/UnitTest/include/TestResult.h, Logical/UnitTest/Libraries/UnitTest/include/TestCase.h, Logical/UnitTest/Samples/Tests_Program/SPLMyCalc/SPLMyCalc.var, Logical/UnitTest/Samples/Tests_Program/Tests_MyCalcLib_C/SPL_CalcTest/testSuite.c, Logical/UnitTest/Samples/Tests_Program/Tests_MyCalcLib_C/SPL_CalcTest/autoGeneratedFile.c, Logical/UnitTest/Samples/Tests_Program/Tests_MyCalcLib_C/SPL_CalcTest/testSet_MyCalcLib_Addition.c, Logical/UnitTest/Samples/Tests_Program/Tests_MyCalcLib_C/SPL_CalcTest/testSet_MyCalcLib_Mult_Div.c, Logical/UnitTest/Samples/Tests_Program/Tests_MyCalcLib_C/SPL_CalcTest_Variants/variables.var, Logical/UnitTest/Samples/Tests_Program/Tests_MyCalcLib_C/SPL_CalcTest_Variants/testSet_MyCalcLib_Subtraction.c, Logical/UnitTest/Samples/Tests_Program/Tests_MyCalcLib_C/SPL_CalcTest_Variants/testSet_MyCalcLib_Subtraction_variantA.c, Logical/UnitTest/Samples/Framework_Extension_With_Custom_Asserts/LibAssert1/LibAssert1_ThresholdAssert.h, Logical/UnitTest/Samples/Framework_Extension_With_Custom_Asserts/LibAssert1/LibAssert1_REAL_ArrayAsserts.h, Logical/UnitTest/Samples/Framework_Extension_With_Custom_Asserts/LibAssert1/LibAssert1_REAL_ArrayAsserts.c, Logical/UnitTest/Samples/Framework_Extension_With_Custom_Asserts/SPL_AssertsEx/testSuite.var, Logical/UnitTest/Samples/Framework_Extension_With_Custom_Asserts/SPL_AssertsEx/autoGeneratedFile.c, Logical/UnitTest/Samples/Framework_Extension_With_Custom_Asserts/SPL_AssertsEx/testSet_AssertsExt.c, Logical/UnitTest/Samples/Framework_Features/SPL_Asserts/testSuite.var, Logical/UnitTest/Samples/Framework_Features/SPL_Asserts/testSuite.c, Logical/UnitTest/Samples/Framework_Features/SPL_Asserts/autoGeneratedFile.c, Logical/UnitTest/Samples/Framework_Features/SPL_Asserts/varAsserts.var, Logical/UnitTest/Samples/Framework_Features/SPL_Asserts/testSet_Asserts.c, Logical/UnitTest/Samples/Framework_Features/SPL_Behavior/testSuite.c, Logical/UnitTest/Samples/Framework_Features/SPL_Behavior/iPrototypes.h, Logical/UnitTest/Samples/Framework_Features/SPL_Behavior/iHelperFunction.h, Logical/UnitTest/Samples/Framework_Features/SPL_Behavior/controlFlowVariables.var, Logical/UnitTest/Samples/Framework_Features/SPL_Behavior/ControlFlow/test_SetTestCases.c, Logical/UnitTest/Samples/Framework_Features/SPL_Behavior/ControlFlow/test_SetTestCases_SetSetup_SetTeardown.c, Logical/UnitTest/Samples/Framework_Features/SPL_Behavior/ControlFlow/test_SetTestCases_TestSetup_TestTeardown.c, Logical/UnitTest/Samples/Framework_Features/SPL_Behavior/TestBusy_AsyncronousVariables.var, Logical/UnitTest/Samples/Framework_Features/SPL_Behavior/TestBusy_Asyncronous/TestBusy_Asyncronous.c, Logical/UnitTest/Samples/Framework_Features/SPL_Behavior/TestBusy_Asyncronous/TestBusy_Asyncronous_with_CyclicSet.c, Logical/UnitTest/Templates/HelperTool_Supported/utTemplate_automated/testSuite.c, Logical/UnitTest/Templates/HelperTool_Supported/utTemplate_automated/autoGeneratedFile.c, Logical/UnitTest/Templates/NoToolSupport/utTemplate_manual/testSuite.c, Logical/UnitTest/Templates/NoToolSupport/utTemplate_manual/FixtureOfTestSets.c, Logical/UnitTest/Templates/NoToolSupport/TestSet_Templates/Set_Testcases.c, Logical/UnitTest/Audit/AuditTest/autoGeneratedFile.c, Logical/UnitTest/Common/CommonUT/CommonTypes.typ, Logical/UnitTest/AppAxis_1/AppAxisUnitTest/autoGeneratedFile.c, Logical/UnitTest/Usb, Logical/UnitTest/Common/CommonUT/CommonTypes.typ, Logical/UnitTest/Report/ReportUnitTest/variables.var, Logical/UnitTest/Common/CommonUT/CommonTypes.typ, Logical/UnitTestVC4/Common/CommonUT/CommonVariables.var, Logical/UnitTestVC4/Audit/AuditTest/Types.typ, Logical/UnitTestVC4/Common/CommonUT/CommonVariables.var, Logical/UnitTestVC4/Backup/BackupUnitTest/autoGeneratedFile.c, Logical/UnitTestVC4/Common/CommonUT/CommonVariables.var, Logical/UnitTestVC4/Common/CommonUT/CommonVariables.var, Logical/UnitTestVC4/File/FileUnitTest/autoGeneratedFile.c, Logical/UnitTestVC4/Usb, Logical/UnitTest/Common/CommonUT/CommonTypes.typ, Logical/UnitTestVC4/Common/CommonUT/CommonVariables.var, Logical/UnitTestVC4/Recipe/RecipeMgrUnitTest/autoGeneratedFile.c, Logical/UnitTestVC4/UserX/UserXUnitTest/autoGeneratedFile.c, Logical/UnitTestVC4/UserX/UserXUnitTest/Set_UserXMgr.c, Logical/UnitTestVC4/Common/CommonUT/CommonVariables.var, Logical/UnitTestVC4/Report/ReportUnitTest/testSuite.c, Logical/UnitTestVC4/Report/ReportUnitTest/autoGeneratedFile.c, Logical/UnitTestVC4/Common/CommonUT/CommonVariables.var, Logical/UnitTestVC4/Common/CommonUT/CommonVariables.var, Logical/UnitTestVC4/Common/CommonUT/autoGeneratedFile.c
